{attribute addProperty BoxType "EL1258-0000-0017"}
{attribute addProperty Id "CtrlAT %Q*Ctrl_2D553DD1324"}
{attribute addProperty CRC "267920111"}
{attribute addProperty SizeInBites "32"}
{attribute addProperty SizeInBytes "4"}
TYPE MTI_Outputs_Channel_0FF822EF :
STRUCT
	{attribute addProperty Name "Ctrl"}
	Ctrl AT %Q* : Ctrl_2D553DD1;
END_STRUCT
END_TYPE

(* stored: Version 1.2.0.0, ProductVersion 3.1.4024.9
   DUT MTI_Outputs_Channel_0FF822EF: Id {3afbff61-58ef-4db7-bd8e-97ea61c0e73b} *)
